(* Logix 5000 project; controller cal1632 1756-L62 rev 16.20; software revision 16.05; part 19 of 57 *)
(* tags used below, declared in another part *)
   FAULT : BOOL;
   HMI : BOOL;
   p01_sys_scp : SYS_SCP;
   p01r09_pb_global_reset : BOOL;
   p13_ai_exhaust_amps : REAL;
   p13_ai_exhaust_hz : REAL;
   p13_ai_exhaust_pct : REAL;
   p13_ai_exhaust_rpm : REAL;
   p13_ai_recirc_amps : REAL;
   p13_ai_recirc_hz : REAL;
   p13_ai_recirc_pct : REAL;
   p13_ai_recirc_rpm : REAL;
   p13_ai_tc01 : REAL;
   p13_ai_tc02 : REAL;
   p13_ao_cv : REAL;
   p13_ao_exhaust_selected_speed : REAL;
   p13_ao_recirc_selected_speed : REAL;
   p13_di_door_open : BOOL;
   p13_di_exh : acs800_di_normal;
   p13_di_exh_fan_mtr_ts : BOOL;
   p13_di_exh_flow_ok : BOOL;
   p13_di_filter_clean : BOOL;
   p13_di_recirc : acs800_di_normal;
   p13_di_recirc_fan_mtr_ts : BOOL;
   p13_di_recirc_flow_ok : BOOL;
   p13_di_tc01_bo : BOOL;
   p13_di_tc02_bo : BOOL;
   p13_dint_to_hmi : DINT[16];
   p13_do_exh : acs800_do_normal;
   p13_do_recirc : acs800_do_normal;
   p13_exhaust_input_max : REAL;
   p13_exhaust_input_min : REAL;
   p13_exhaust_output_max : REAL;
   p13_exhaust_output_min : REAL;
   p13_hc_input_max : REAL;
   p13_hc_input_min : REAL;
   p13_hc_output_max : REAL;
   p13_hc_output_min : REAL;
   p13_param_fast_to_soak : REAL;
   p13_param_lfl_hhl : REAL;
   p13_param_lfl_hl : REAL;
   p13_param_pid1_ff : REAL;
   p13_param_pid1_kd : REAL;
   p13_param_pid1_ki : REAL;
   p13_param_pid1_kp : REAL;
   p13_param_pid2_ff : REAL;
   p13_param_pid2_kd : REAL;
   p13_param_pid2_ki : REAL;
   p13_param_pid2_kp : REAL;
   p13_param_shutdown_temp : REAL;
   p13_param_soak_to_fast : REAL;
   p13_param_tc01_dev : REAL;
   p13_param_tc01_hl : REAL;
   p13_param_tc01z : REAL;
   p13_param_tc02z : REAL;
   p13_param_zone_pressure : REAL;
   p13_real_to_hmi : REAL[112];
   p13_recirc_input_max : REAL;
   p13_recirc_input_min : REAL;
   p13_recirc_output_max : REAL;
   p13_recirc_output_min : REAL;
   p13r04 : routine;
   p13r04_timer_fault : TIMER[4];
   p13r04_timer_warning : TIMER[4];
   p13r05 : routine;
   p13r05_exh_status : DINT;
   p13r05_recirc_status : DINT;
   p13r05_temp_ctl_status : DINT;
   p13r05_timer_fault : TIMER[4];
   p13r05_timer_warning : TIMER[4];
   p13r06 : routine;
   p13r06_timer_fault : TIMER[4];
   p13r06_timer_warning : TIMER[4];
   p13r20_state : DINT;
   p13r20_status : DINT;
   p13r30 : routine;
   p13r30_cv_man_sp : REAL;
   p13r30_permissive_run : BOOL;
   p13r30_pid_temp_pv : REAL;
   p13r30_pid_temp_sp : REAL;
   p13r30_request_cool : BOOL;
   p13r30_request_manual : BOOL;
   p13r30_vfds_ready : BOOL;
   p13r31 : routine;
   p13r31_request_auto_run : BOOL;
   p13r31_request_auto_stop : BOOL;
   p13r31_vfd_stopped : BOOL;
   p13r32 : routine;
   p13r32_request_auto_run : BOOL;
   p13r32_request_auto_stop : BOOL;
   p13r32_vfd_stopped : BOOL;
(* P13_Zone_3, continued *)

ROUTINE R04_Output   (* ladder *)
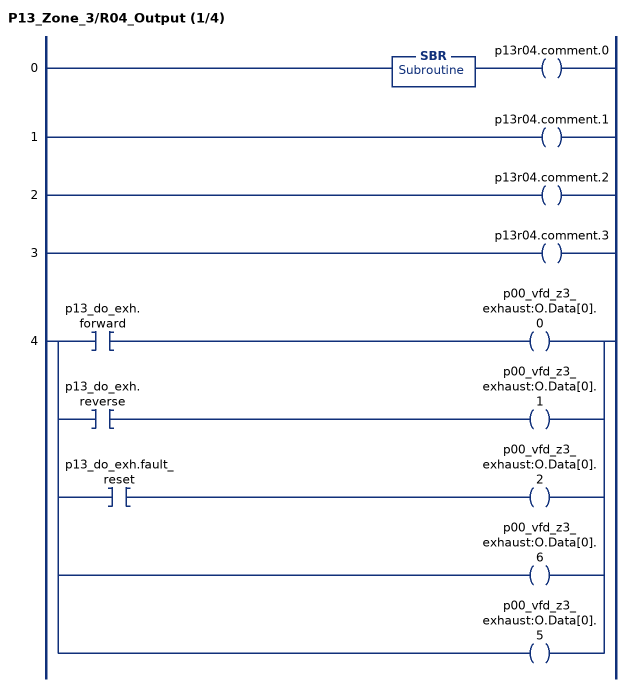
   0: SBR()OTE(p13r04.comment.0);
   1: OTE(p13r04.comment.1);
   2: OTE(p13r04.comment.2);
   3: OTE(p13r04.comment.3);
   4: [XIC(p13_do_exh.forward) OTE(p00_vfd_z3_exhaust:O.Data[0].0) ,XIC(p13_do_exh.reverse) OTE(p00_vfd_z3_exhaust:O.Data[0].1) ,XIC(p13_do_exh.fault_reset) OTE(p00_vfd_z3_exhaust:O.Data[0].2) ,OTE(p00_vfd_z3_exhaust:O.Data[0].6) ,OTE(p00_vfd_z3_exhaust:O.Data[0].5) ];
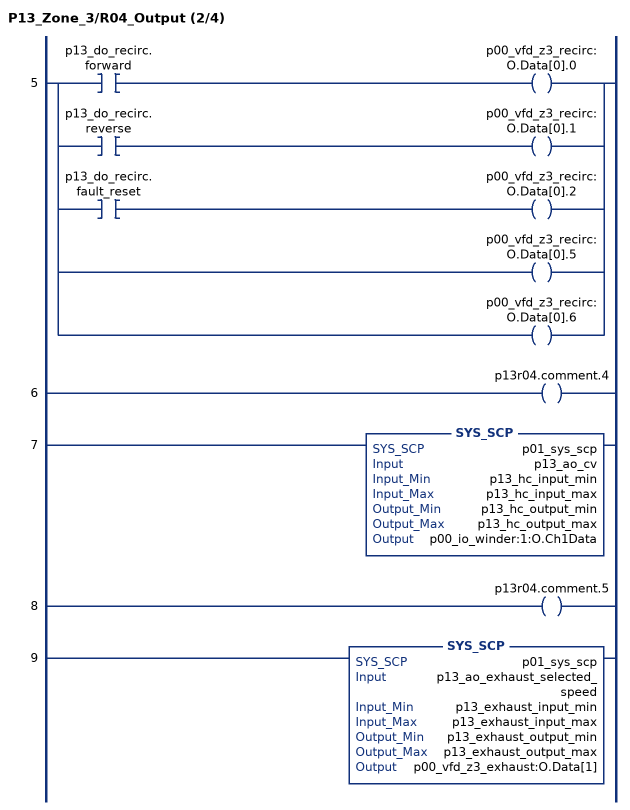
   5: [XIC(p13_do_recirc.forward) OTE(p00_vfd_z3_recirc:O.Data[0].0) ,XIC(p13_do_recirc.reverse) OTE(p00_vfd_z3_recirc:O.Data[0].1) ,XIC(p13_do_recirc.fault_reset) OTE(p00_vfd_z3_recirc:O.Data[0].2) ,OTE(p00_vfd_z3_recirc:O.Data[0].5) ,OTE(p00_vfd_z3_recirc:O.Data[0].6) ];
   6: OTE(p13r04.comment.4);
   7: SYS_SCP(p01_sys_scp,p13_ao_cv,p13_hc_input_min,p13_hc_input_max,p13_hc_output_min,p13_hc_output_max,p00_io_winder:1:O.Ch1Data);
   8: OTE(p13r04.comment.5);
   9: SYS_SCP(p01_sys_scp,p13_ao_exhaust_selected_speed,p13_exhaust_input_min,p13_exhaust_input_max,p13_exhaust_output_min,p13_exhaust_output_max,p00_vfd_z3_exhaust:O.Data[1]);
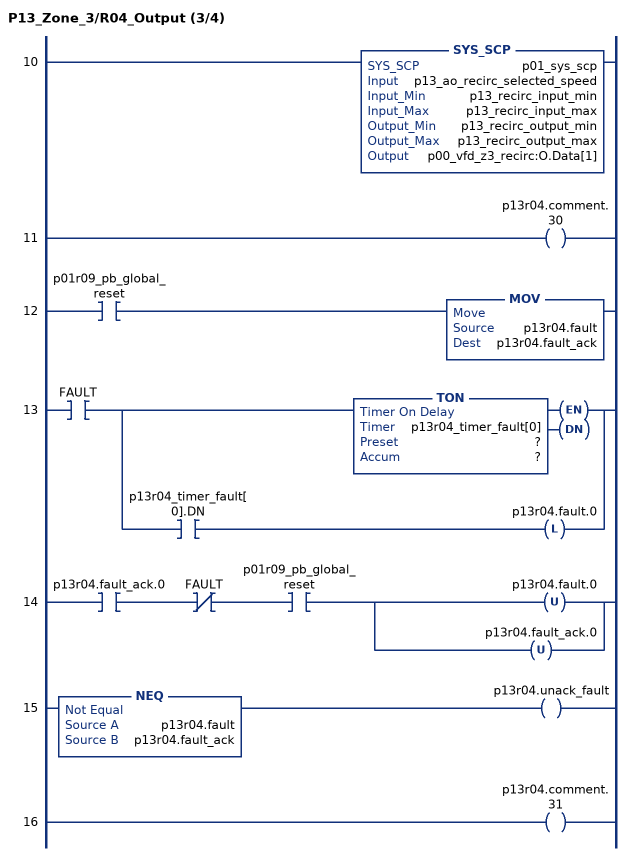
   10: SYS_SCP(p01_sys_scp,p13_ao_recirc_selected_speed,p13_recirc_input_min,p13_recirc_input_max,p13_recirc_output_min,p13_recirc_output_max,p00_vfd_z3_recirc:O.Data[1]);
   11: OTE(p13r04.comment.30);
   12: XIC(p01r09_pb_global_reset)MOV(p13r04.fault,p13r04.fault_ack);
   13: XIC(FAULT)[TON(p13r04_timer_fault[0],?,?) ,XIC(p13r04_timer_fault[0].DN) OTL(p13r04.fault.0) ];
   14: XIC(p13r04.fault_ack.0)XIO(FAULT)XIC(p01r09_pb_global_reset)[OTU(p13r04.fault.0) ,OTU(p13r04.fault_ack.0) ];
   15: NEQ(p13r04.fault,p13r04.fault_ack)OTE(p13r04.unack_fault);
   16: OTE(p13r04.comment.31);
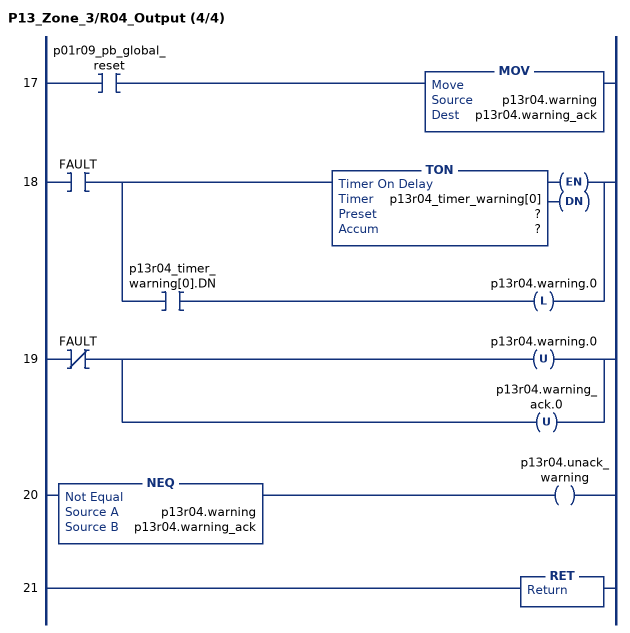
   17: XIC(p01r09_pb_global_reset)MOV(p13r04.warning,p13r04.warning_ack);
   18: XIC(FAULT)[TON(p13r04_timer_warning[0],?,?) ,XIC(p13r04_timer_warning[0].DN) OTL(p13r04.warning.0) ];
   19: XIO(FAULT)[OTU(p13r04.warning.0) ,OTU(p13r04.warning_ack.0) ];
   20: NEQ(p13r04.warning,p13r04.warning_ack)OTE(p13r04.unack_warning);
   21: RET();
END_ROUTINE

ROUTINE R05_Dint_to_HMI   (* ladder *)
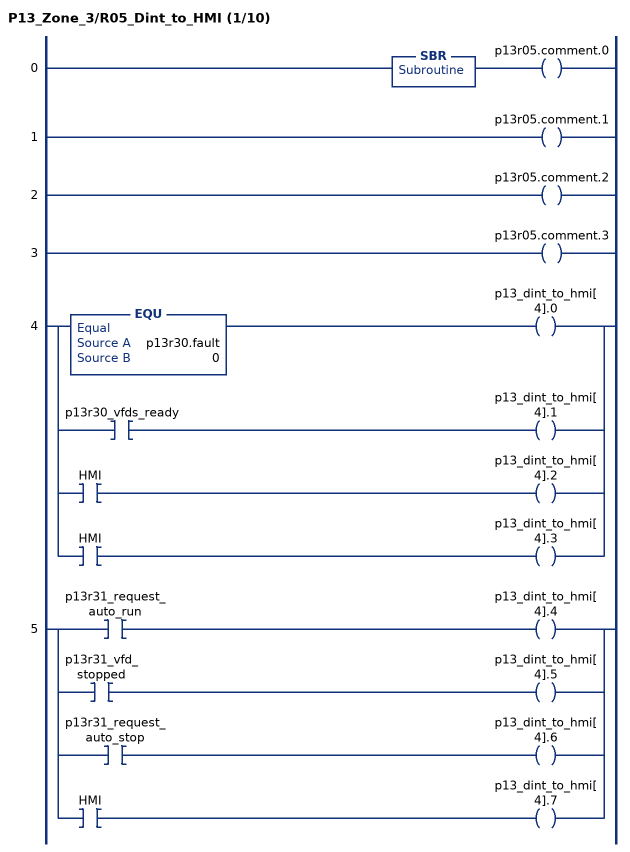
   0: SBR()OTE(p13r05.comment.0);
   1: OTE(p13r05.comment.1);
   2: OTE(p13r05.comment.2);
   3: OTE(p13r05.comment.3);
   4: [EQU(p13r30.fault,0) OTE(p13_dint_to_hmi[4].0) ,XIC(p13r30_vfds_ready) OTE(p13_dint_to_hmi[4].1) ,XIC(HMI) OTE(p13_dint_to_hmi[4].2) ,XIC(HMI) OTE(p13_dint_to_hmi[4].3) ];
   5: [XIC(p13r31_request_auto_run) OTE(p13_dint_to_hmi[4].4) ,XIC(p13r31_vfd_stopped) OTE(p13_dint_to_hmi[4].5) ,XIC(p13r31_request_auto_stop) OTE(p13_dint_to_hmi[4].6) ,XIC(HMI) OTE(p13_dint_to_hmi[4].7) ];
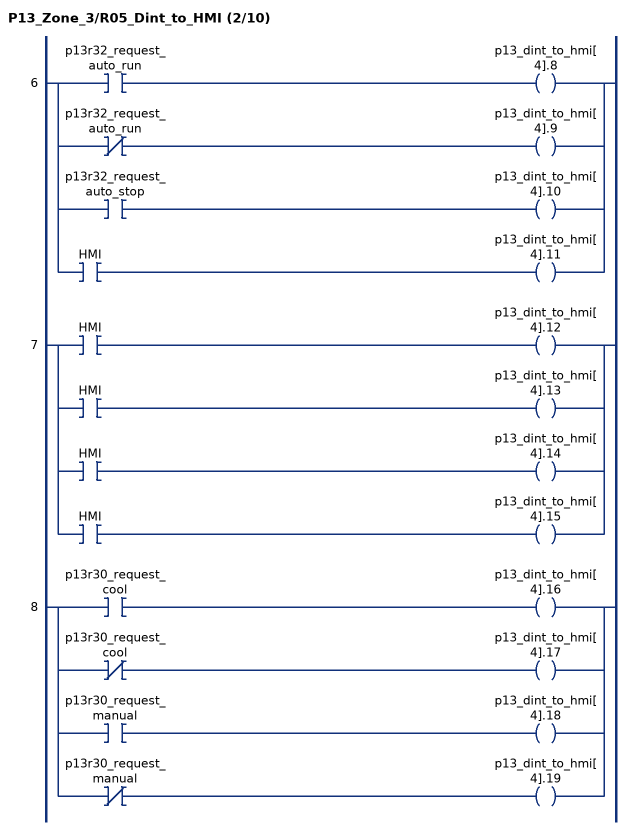
   6: [XIC(p13r32_request_auto_run) OTE(p13_dint_to_hmi[4].8) ,XIO(p13r32_request_auto_run) OTE(p13_dint_to_hmi[4].9) ,XIC(p13r32_request_auto_stop) OTE(p13_dint_to_hmi[4].10) ,XIC(HMI) OTE(p13_dint_to_hmi[4].11) ];
   7: [XIC(HMI) OTE(p13_dint_to_hmi[4].12) ,XIC(HMI) OTE(p13_dint_to_hmi[4].13) ,XIC(HMI) OTE(p13_dint_to_hmi[4].14) ,XIC(HMI) OTE(p13_dint_to_hmi[4].15) ];
   8: [XIC(p13r30_request_cool) OTE(p13_dint_to_hmi[4].16) ,XIO(p13r30_request_cool) OTE(p13_dint_to_hmi[4].17) ,XIC(p13r30_request_manual) OTE(p13_dint_to_hmi[4].18) ,XIO(p13r30_request_manual) OTE(p13_dint_to_hmi[4].19) ];
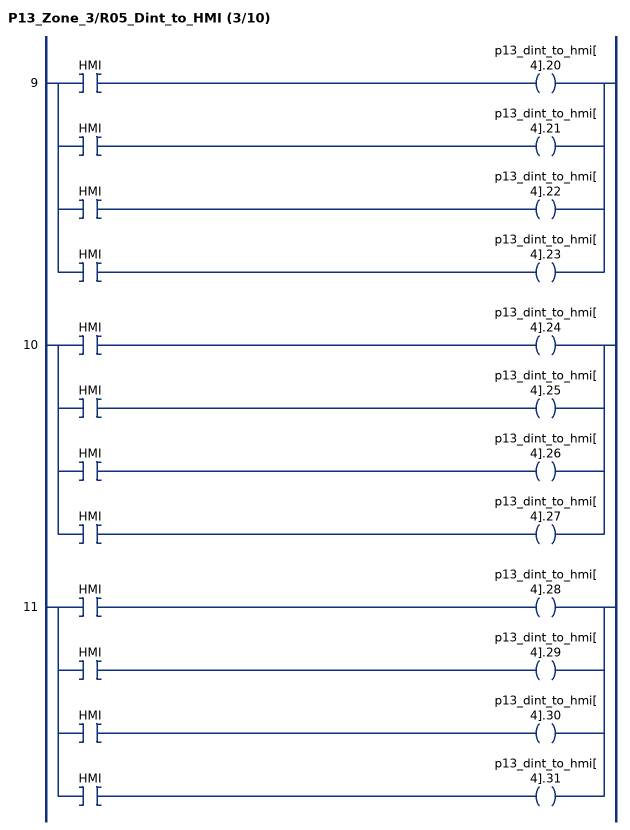
   9: [XIC(HMI) OTE(p13_dint_to_hmi[4].20) ,XIC(HMI) OTE(p13_dint_to_hmi[4].21) ,XIC(HMI) OTE(p13_dint_to_hmi[4].22) ,XIC(HMI) OTE(p13_dint_to_hmi[4].23) ];
   10: [XIC(HMI) OTE(p13_dint_to_hmi[4].24) ,XIC(HMI) OTE(p13_dint_to_hmi[4].25) ,XIC(HMI) OTE(p13_dint_to_hmi[4].26) ,XIC(HMI) OTE(p13_dint_to_hmi[4].27) ];
   11: [XIC(HMI) OTE(p13_dint_to_hmi[4].28) ,XIC(HMI) OTE(p13_dint_to_hmi[4].29) ,XIC(HMI) OTE(p13_dint_to_hmi[4].30) ,XIC(HMI) OTE(p13_dint_to_hmi[4].31) ];
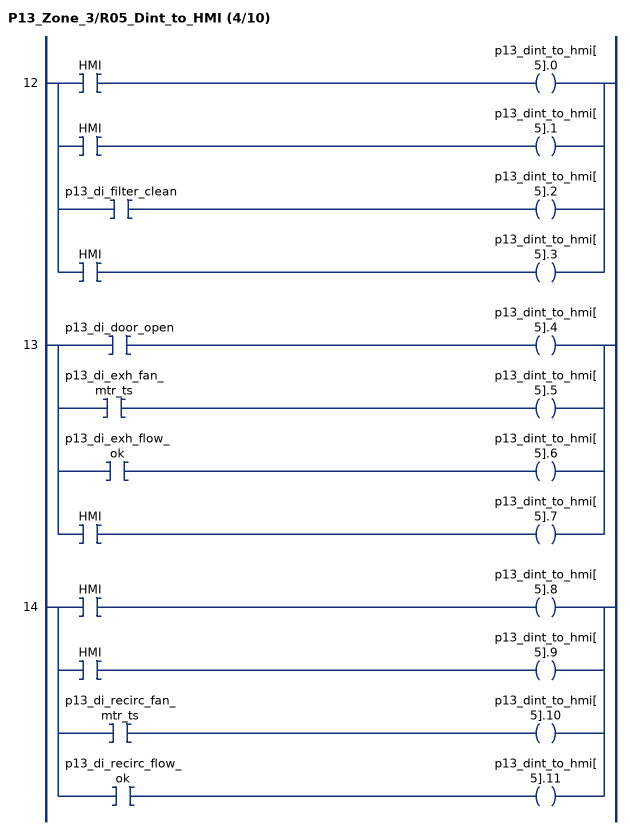
   12: [XIC(HMI) OTE(p13_dint_to_hmi[5].0) ,XIC(HMI) OTE(p13_dint_to_hmi[5].1) ,XIC(p13_di_filter_clean) OTE(p13_dint_to_hmi[5].2) ,XIC(HMI) OTE(p13_dint_to_hmi[5].3) ];
   13: [XIC(p13_di_door_open) OTE(p13_dint_to_hmi[5].4) ,XIC(p13_di_exh_fan_mtr_ts) OTE(p13_dint_to_hmi[5].5) ,XIC(p13_di_exh_flow_ok) OTE(p13_dint_to_hmi[5].6) ,XIC(HMI) OTE(p13_dint_to_hmi[5].7) ];
   14: [XIC(HMI) OTE(p13_dint_to_hmi[5].8) ,XIC(HMI) OTE(p13_dint_to_hmi[5].9) ,XIC(p13_di_recirc_fan_mtr_ts) OTE(p13_dint_to_hmi[5].10) ,XIC(p13_di_recirc_flow_ok) OTE(p13_dint_to_hmi[5].11) ];
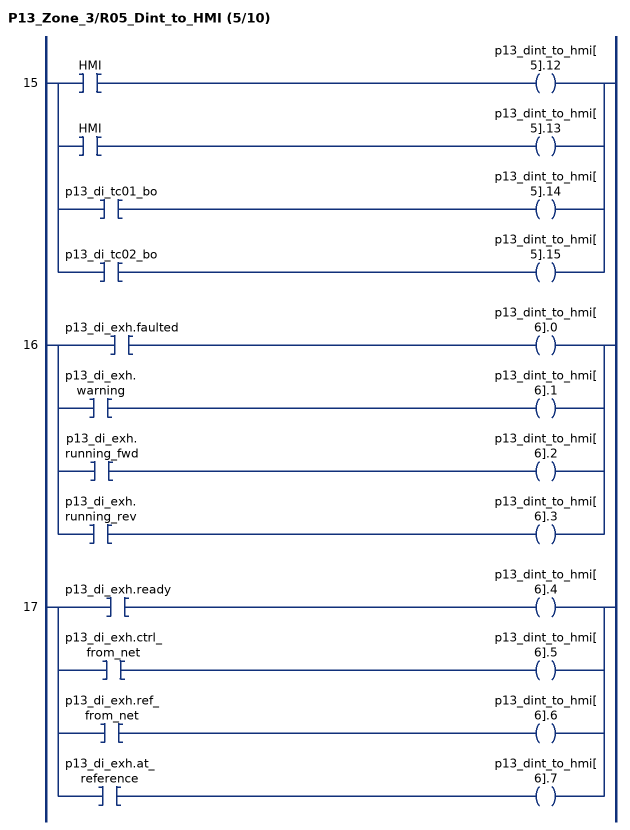
   15: [XIC(HMI) OTE(p13_dint_to_hmi[5].12) ,XIC(HMI) OTE(p13_dint_to_hmi[5].13) ,XIC(p13_di_tc01_bo) OTE(p13_dint_to_hmi[5].14) ,XIC(p13_di_tc02_bo) OTE(p13_dint_to_hmi[5].15) ];
   16: [XIC(p13_di_exh.faulted) OTE(p13_dint_to_hmi[6].0) ,XIC(p13_di_exh.warning) OTE(p13_dint_to_hmi[6].1) ,XIC(p13_di_exh.running_fwd) OTE(p13_dint_to_hmi[6].2) ,XIC(p13_di_exh.running_rev) OTE(p13_dint_to_hmi[6].3) ];
   17: [XIC(p13_di_exh.ready) OTE(p13_dint_to_hmi[6].4) ,XIC(p13_di_exh.ctrl_from_net) OTE(p13_dint_to_hmi[6].5) ,XIC(p13_di_exh.ref_from_net) OTE(p13_dint_to_hmi[6].6) ,XIC(p13_di_exh.at_reference) OTE(p13_dint_to_hmi[6].7) ];
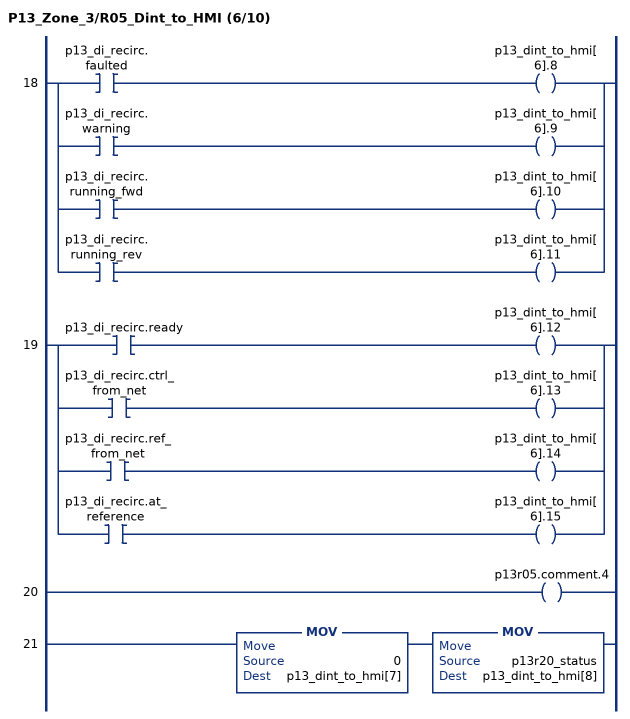
   18: [XIC(p13_di_recirc.faulted) OTE(p13_dint_to_hmi[6].8) ,XIC(p13_di_recirc.warning) OTE(p13_dint_to_hmi[6].9) ,XIC(p13_di_recirc.running_fwd) OTE(p13_dint_to_hmi[6].10) ,XIC(p13_di_recirc.running_rev) OTE(p13_dint_to_hmi[6].11) ];
   19: [XIC(p13_di_recirc.ready) OTE(p13_dint_to_hmi[6].12) ,XIC(p13_di_recirc.ctrl_from_net) OTE(p13_dint_to_hmi[6].13) ,XIC(p13_di_recirc.ref_from_net) OTE(p13_dint_to_hmi[6].14) ,XIC(p13_di_recirc.at_reference) OTE(p13_dint_to_hmi[6].15) ];
   20: OTE(p13r05.comment.4);
   21: MOV(0,p13_dint_to_hmi[7])MOV(p13r20_status,p13_dint_to_hmi[8]);
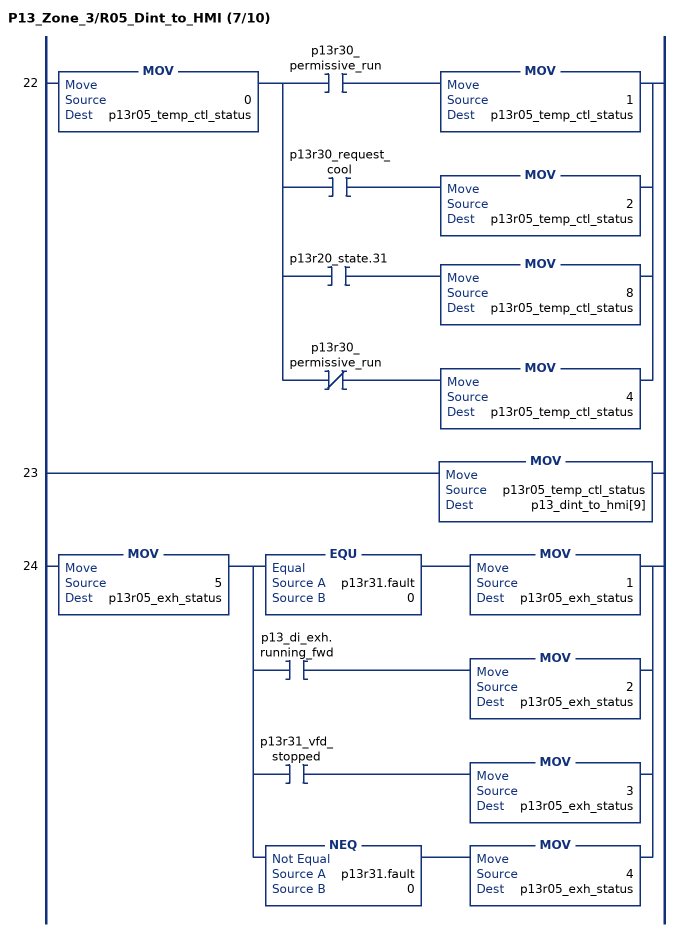
   22: MOV(0,p13r05_temp_ctl_status)[XIC(p13r30_permissive_run) MOV(1,p13r05_temp_ctl_status) ,XIC(p13r30_request_cool) MOV(2,p13r05_temp_ctl_status) ,XIC(p13r20_state.31) MOV(8,p13r05_temp_ctl_status) ,XIO(p13r30_permissive_run) MOV(4,p13r05_temp_ctl_status) ];
   23: MOV(p13r05_temp_ctl_status,p13_dint_to_hmi[9]);
   24: MOV(5,p13r05_exh_status)[EQU(p13r31.fault,0) MOV(1,p13r05_exh_status) ,XIC(p13_di_exh.running_fwd) MOV(2,p13r05_exh_status) ,XIC(p13r31_vfd_stopped) MOV(3,p13r05_exh_status) ,NEQ(p13r31.fault,0) MOV(4,p13r05_exh_status) ];
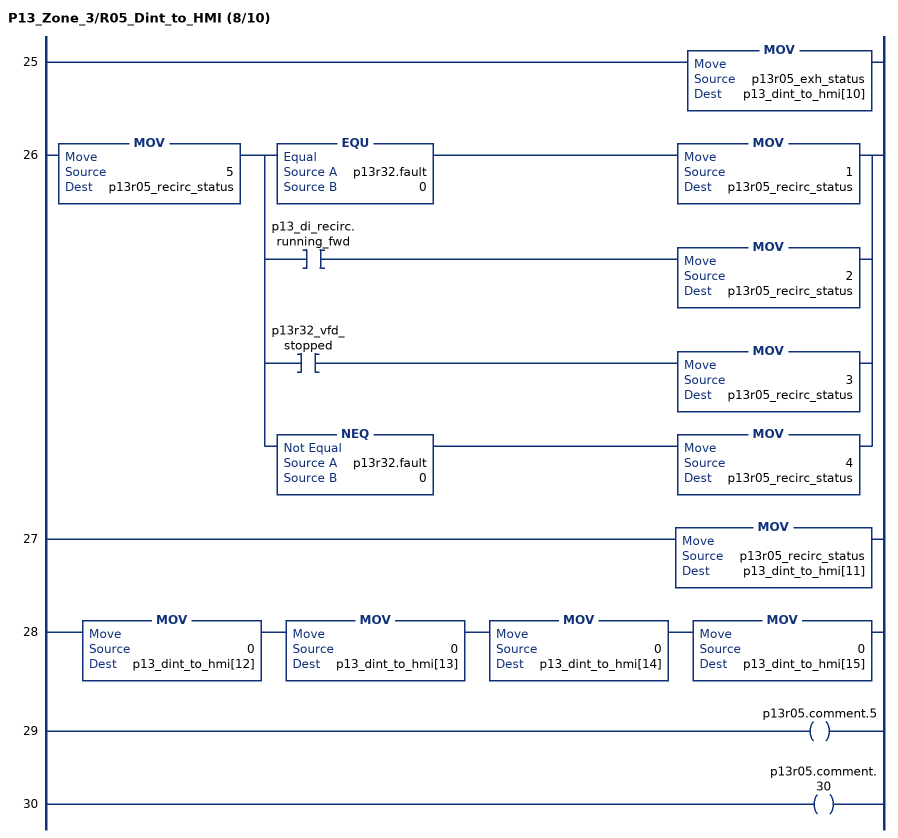
   25: MOV(p13r05_exh_status,p13_dint_to_hmi[10]);
   26: MOV(5,p13r05_recirc_status)[EQU(p13r32.fault,0) MOV(1,p13r05_recirc_status) ,XIC(p13_di_recirc.running_fwd) MOV(2,p13r05_recirc_status) ,XIC(p13r32_vfd_stopped) MOV(3,p13r05_recirc_status) ,NEQ(p13r32.fault,0) MOV(4,p13r05_recirc_status) ];
   27: MOV(p13r05_recirc_status,p13_dint_to_hmi[11]);
   28: MOV(0,p13_dint_to_hmi[12])MOV(0,p13_dint_to_hmi[13])MOV(0,p13_dint_to_hmi[14])MOV(0,p13_dint_to_hmi[15]);
   29: OTE(p13r05.comment.5);
   30: OTE(p13r05.comment.30);
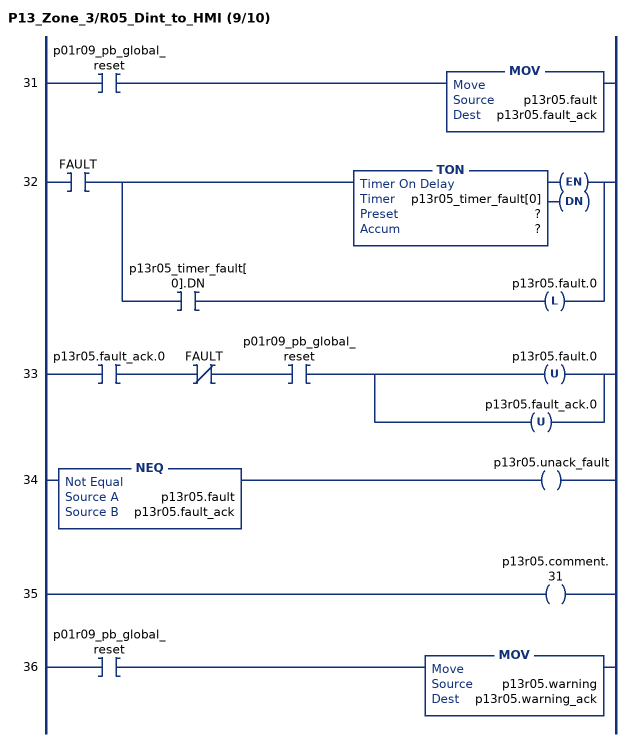
   31: XIC(p01r09_pb_global_reset)MOV(p13r05.fault,p13r05.fault_ack);
   32: XIC(FAULT)[TON(p13r05_timer_fault[0],?,?) ,XIC(p13r05_timer_fault[0].DN) OTL(p13r05.fault.0) ];
   33: XIC(p13r05.fault_ack.0)XIO(FAULT)XIC(p01r09_pb_global_reset)[OTU(p13r05.fault.0) ,OTU(p13r05.fault_ack.0) ];
   34: NEQ(p13r05.fault,p13r05.fault_ack)OTE(p13r05.unack_fault);
   35: OTE(p13r05.comment.31);
   36: XIC(p01r09_pb_global_reset)MOV(p13r05.warning,p13r05.warning_ack);
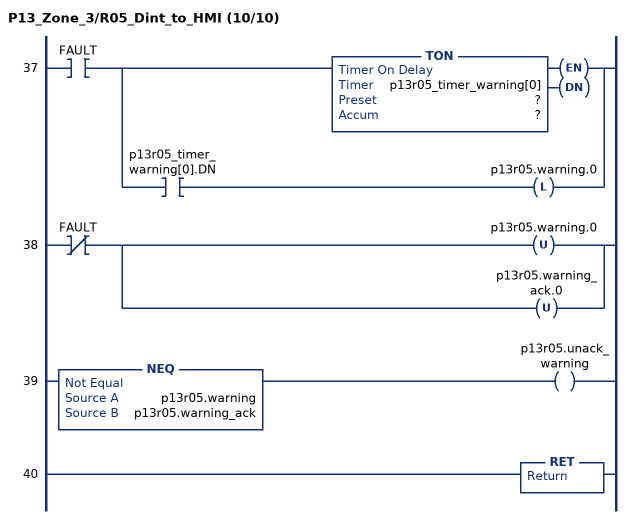
   37: XIC(FAULT)[TON(p13r05_timer_warning[0],?,?) ,XIC(p13r05_timer_warning[0].DN) OTL(p13r05.warning.0) ];
   38: XIO(FAULT)[OTU(p13r05.warning.0) ,OTU(p13r05.warning_ack.0) ];
   39: NEQ(p13r05.warning,p13r05.warning_ack)OTE(p13r05.unack_warning);
   40: RET();
END_ROUTINE

ROUTINE R06_Real_to_HMI   (* ladder *)
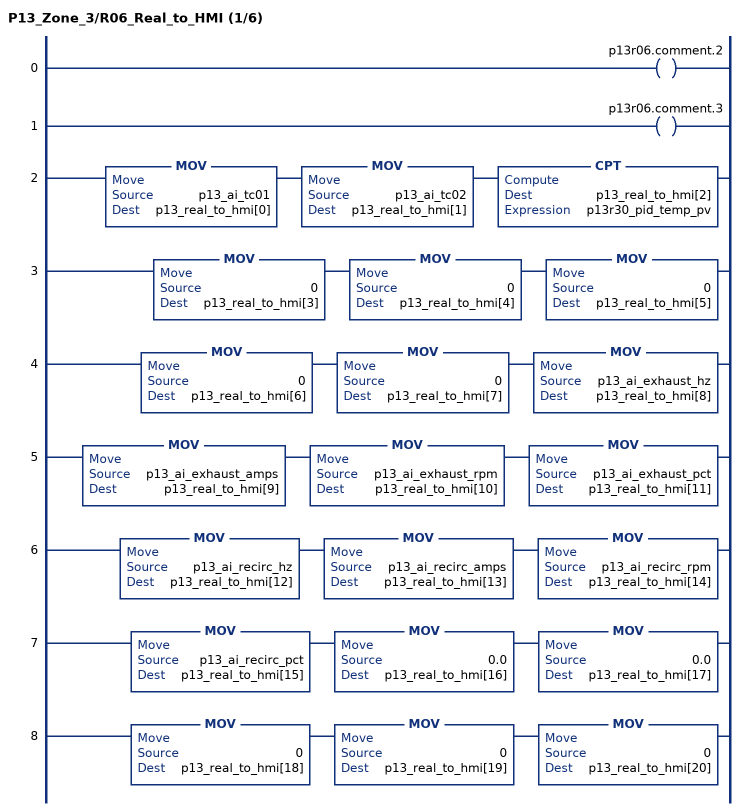
   0: OTE(p13r06.comment.2);
   1: OTE(p13r06.comment.3);
   2: MOV(p13_ai_tc01,p13_real_to_hmi[0])MOV(p13_ai_tc02,p13_real_to_hmi[1])CPT(p13_real_to_hmi[2],p13r30_pid_temp_pv);
   3: MOV(0,p13_real_to_hmi[3])MOV(0,p13_real_to_hmi[4])MOV(0,p13_real_to_hmi[5]);
   4: MOV(0,p13_real_to_hmi[6])MOV(0,p13_real_to_hmi[7])MOV(p13_ai_exhaust_hz,p13_real_to_hmi[8]);
   5: MOV(p13_ai_exhaust_amps,p13_real_to_hmi[9])MOV(p13_ai_exhaust_rpm,p13_real_to_hmi[10])MOV(p13_ai_exhaust_pct,p13_real_to_hmi[11]);
   6: MOV(p13_ai_recirc_hz,p13_real_to_hmi[12])MOV(p13_ai_recirc_amps,p13_real_to_hmi[13])MOV(p13_ai_recirc_rpm,p13_real_to_hmi[14]);
   7: MOV(p13_ai_recirc_pct,p13_real_to_hmi[15])MOV(0.0,p13_real_to_hmi[16])MOV(0.0,p13_real_to_hmi[17]);
   8: MOV(0,p13_real_to_hmi[18])MOV(0,p13_real_to_hmi[19])MOV(0,p13_real_to_hmi[20]);
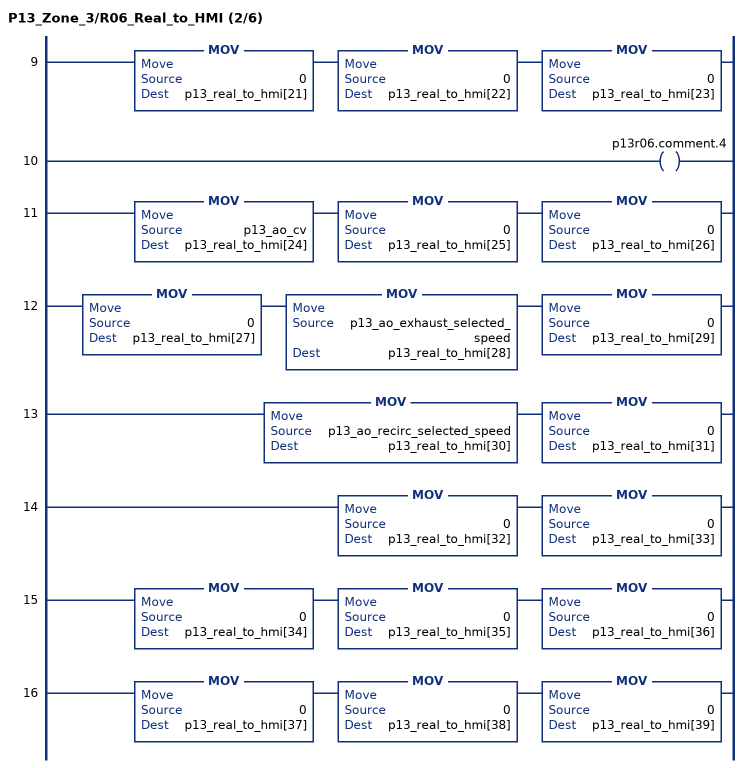
   9: MOV(0,p13_real_to_hmi[21])MOV(0,p13_real_to_hmi[22])MOV(0,p13_real_to_hmi[23]);
   10: OTE(p13r06.comment.4);
   11: MOV(p13_ao_cv,p13_real_to_hmi[24])MOV(0,p13_real_to_hmi[25])MOV(0,p13_real_to_hmi[26]);
   12: MOV(0,p13_real_to_hmi[27])MOV(p13_ao_exhaust_selected_speed,p13_real_to_hmi[28])MOV(0,p13_real_to_hmi[29]);
   13: MOV(p13_ao_recirc_selected_speed,p13_real_to_hmi[30])MOV(0,p13_real_to_hmi[31]);
   14: MOV(0,p13_real_to_hmi[32])MOV(0,p13_real_to_hmi[33]);
   15: MOV(0,p13_real_to_hmi[34])MOV(0,p13_real_to_hmi[35])MOV(0,p13_real_to_hmi[36]);
   16: MOV(0,p13_real_to_hmi[37])MOV(0,p13_real_to_hmi[38])MOV(0,p13_real_to_hmi[39]);
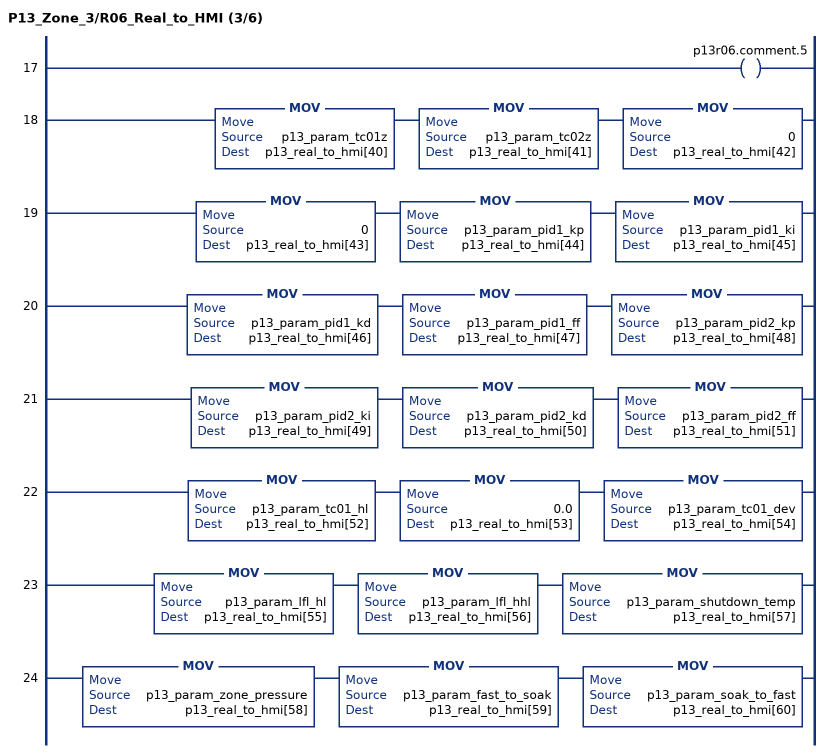
   17: OTE(p13r06.comment.5);
   18: MOV(p13_param_tc01z,p13_real_to_hmi[40])MOV(p13_param_tc02z,p13_real_to_hmi[41])MOV(0,p13_real_to_hmi[42]);
   19: MOV(0,p13_real_to_hmi[43])MOV(p13_param_pid1_kp,p13_real_to_hmi[44])MOV(p13_param_pid1_ki,p13_real_to_hmi[45]);
   20: MOV(p13_param_pid1_kd,p13_real_to_hmi[46])MOV(p13_param_pid1_ff,p13_real_to_hmi[47])MOV(p13_param_pid2_kp,p13_real_to_hmi[48]);
   21: MOV(p13_param_pid2_ki,p13_real_to_hmi[49])MOV(p13_param_pid2_kd,p13_real_to_hmi[50])MOV(p13_param_pid2_ff,p13_real_to_hmi[51]);
   22: MOV(p13_param_tc01_hl,p13_real_to_hmi[52])MOV(0.0,p13_real_to_hmi[53])MOV(p13_param_tc01_dev,p13_real_to_hmi[54]);
   23: MOV(p13_param_lfl_hl,p13_real_to_hmi[55])MOV(p13_param_lfl_hhl,p13_real_to_hmi[56])MOV(p13_param_shutdown_temp,p13_real_to_hmi[57]);
   24: MOV(p13_param_zone_pressure,p13_real_to_hmi[58])MOV(p13_param_fast_to_soak,p13_real_to_hmi[59])MOV(p13_param_soak_to_fast,p13_real_to_hmi[60]);
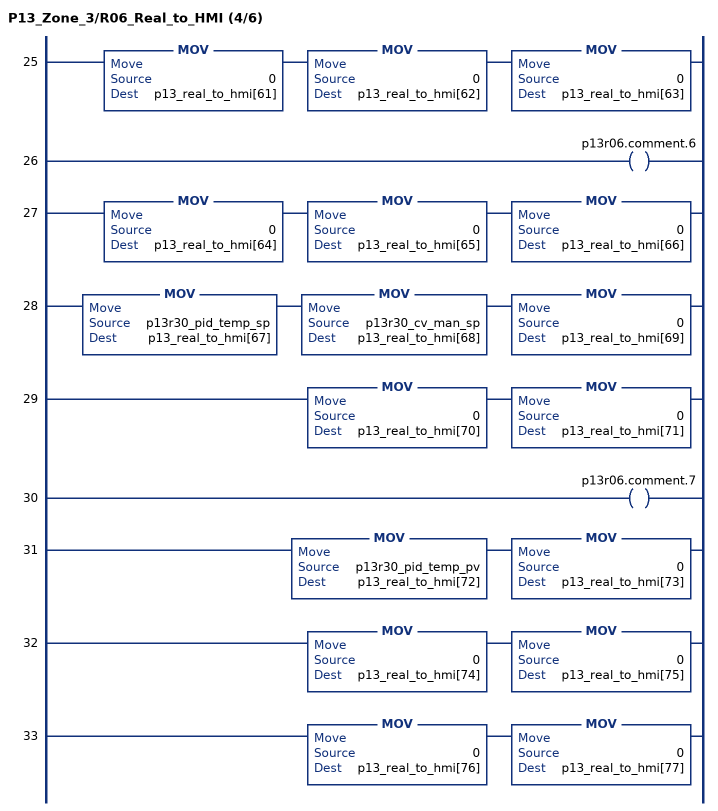
   25: MOV(0,p13_real_to_hmi[61])MOV(0,p13_real_to_hmi[62])MOV(0,p13_real_to_hmi[63]);
   26: OTE(p13r06.comment.6);
   27: MOV(0,p13_real_to_hmi[64])MOV(0,p13_real_to_hmi[65])MOV(0,p13_real_to_hmi[66]);
   28: MOV(p13r30_pid_temp_sp,p13_real_to_hmi[67])MOV(p13r30_cv_man_sp,p13_real_to_hmi[68])MOV(0,p13_real_to_hmi[69]);
   29: MOV(0,p13_real_to_hmi[70])MOV(0,p13_real_to_hmi[71]);
   30: OTE(p13r06.comment.7);
   31: MOV(p13r30_pid_temp_pv,p13_real_to_hmi[72])MOV(0,p13_real_to_hmi[73]);
   32: MOV(0,p13_real_to_hmi[74])MOV(0,p13_real_to_hmi[75]);
   33: MOV(0,p13_real_to_hmi[76])MOV(0,p13_real_to_hmi[77]);
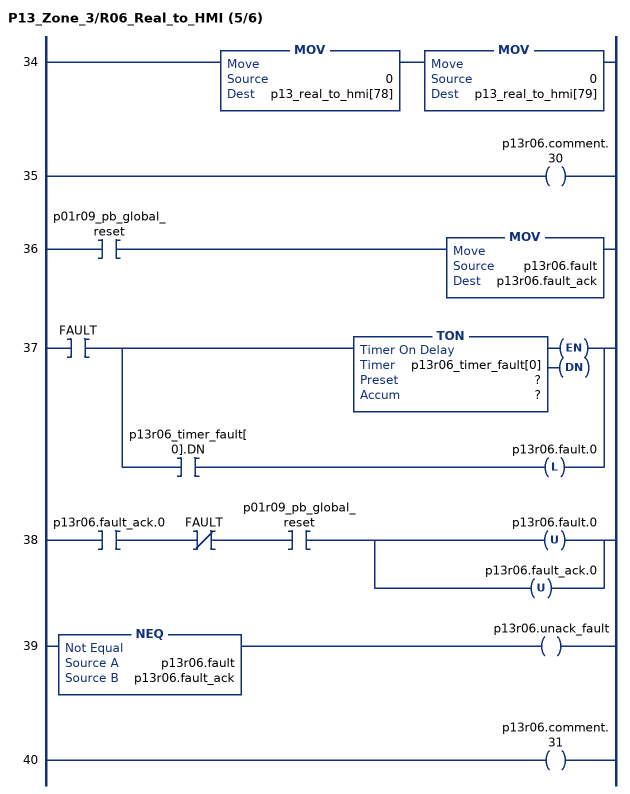
   34: MOV(0,p13_real_to_hmi[78])MOV(0,p13_real_to_hmi[79]);
   35: OTE(p13r06.comment.30);
   36: XIC(p01r09_pb_global_reset)MOV(p13r06.fault,p13r06.fault_ack);
   37: XIC(FAULT)[TON(p13r06_timer_fault[0],?,?) ,XIC(p13r06_timer_fault[0].DN) OTL(p13r06.fault.0) ];
   38: XIC(p13r06.fault_ack.0)XIO(FAULT)XIC(p01r09_pb_global_reset)[OTU(p13r06.fault.0) ,OTU(p13r06.fault_ack.0) ];
   39: NEQ(p13r06.fault,p13r06.fault_ack)OTE(p13r06.unack_fault);
   40: OTE(p13r06.comment.31);
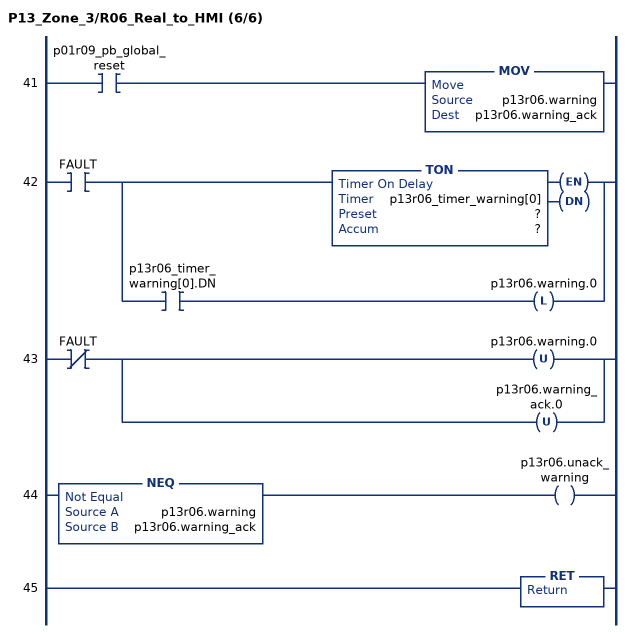
   41: XIC(p01r09_pb_global_reset)MOV(p13r06.warning,p13r06.warning_ack);
   42: XIC(FAULT)[TON(p13r06_timer_warning[0],?,?) ,XIC(p13r06_timer_warning[0].DN) OTL(p13r06.warning.0) ];
   43: XIO(FAULT)[OTU(p13r06.warning.0) ,OTU(p13r06.warning_ack.0) ];
   44: NEQ(p13r06.warning,p13r06.warning_ack)OTE(p13r06.unack_warning);
   45: RET();
END_ROUTINE
